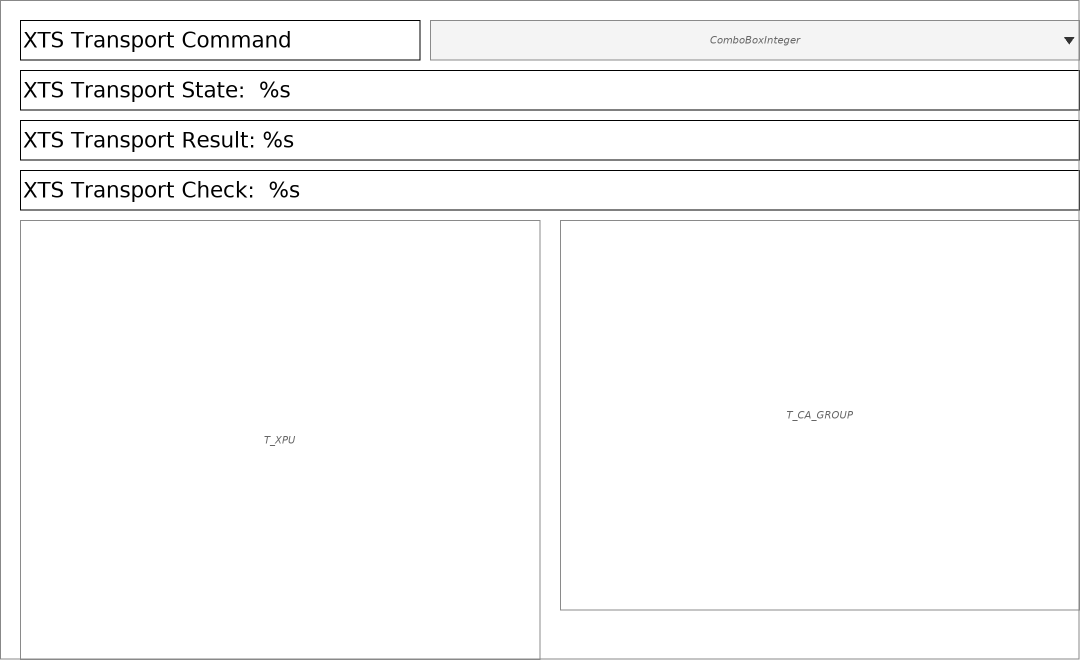
VISUALIZATION XTS_TRANSPORT  // 1080x660
    Rectangle (20,20 400x40), "XTS Transport Command"
    ComboBoxInteger (430,20 650x40), variable: GVL_XTS.XtsTransportCtrl.Cmd, text list: 'TL_E_CTRL_TRANSPORT'
    Rectangle (20,70 1060x40), "XTS Transport State: %s", text variable: VISU_XTS.sTransportState
    Rectangle (20,120 1060x40), "XTS Transport Result: %s", text variable: VISU_XTS.sTransportResult
    Rectangle (20,170 1060x40), "XTS Transport Check: %s", text variable: VISU_XTS.sTransportCheck
    Frame (20,220 520x440)
        shows T_XPU(stXpuState := GVL_XTS.XtsTransportState.XpuState, stXpuInfo := GVL_XTS.XtsTransportState.XpuInfo, stXpuStrings := VISU_XTS.stXpuStrings)
    Frame (560,220 520x390)
        shows T_CA_GROUP(stGroupInfo := GVL_XTS.XtsTransportState.GroupInfo, sGroupState := visu_XTS.sCaGroupState)
END_VISUALIZATION

(* stored: Version 1.1.0.1
   Visu XTS_TRANSPORT: Id {8070c5f6-652f-4902-bd3c-f59a57108227} *)
